  MoveL 7233 to (-64.74, 18.89, -264.72) mm, rotated rx 105.8 ry 33.04 rz 34.05 deg; joints [-10.347, -22.359, 96.233, 141.056, 86.367, 19.409, -475]
  MoveL 7234 to (-64.97, 19.26, -264.23) mm, rotated rx 105.8 ry 33.04 rz 34.05 deg; joints [-10.328, -22.332, 96.216, 141.075, 86.371, 19.399, -475]
  MoveL 7235 to (-64.83, 18.38, -263.37) mm, rotated rx 105.8 ry 33.04 rz 34.05 deg; joints [-10.295, -22.38, 96.234, 141.106, 86.342, 19.41, -475]
  MoveL 7236 to (-64.29, 14.15, -263.37) mm, rotated rx 105.8 ry 33.04 rz 34.05 deg; joints [-10.289, -22.594, 96.267, 141.105, 86.2, 19.523, -475]
  MoveL 7237 to (-64.04, 12.17, -263.31) mm, rotated rx 105.8 ry 33.04 rz 34.05 deg; joints [-10.284, -22.694, 96.282, 141.106, 86.132, 19.576, -475]
  MoveL 7238 to (-63.81, 10.19, -263.16) mm, rotated rx 105.8 ry 33.04 rz 34.05 deg; joints [-10.275, -22.794, 96.296, 141.111, 86.064, 19.628, -475]
  MoveL 7239 to (-63.54, 7.91, -262.96) mm, rotated rx 105.8 ry 33.04 rz 34.05 deg; joints [-10.264, -22.908, 96.312, 141.117, 85.986, 19.687, -475]
  MoveL 7240 to (-63.28, 5.75, -262.75) mm, rotated rx 105.8 ry 33.04 rz 34.05 deg; joints [-10.253, -23.016, 96.327, 141.124, 85.912, 19.743, -475]
  MoveL 7241 to (-63.02, 3.59, -262.65) mm, rotated rx 105.8 ry 33.04 rz 34.05 deg; joints [-10.246, -23.125, 96.342, 141.126, 85.837, 19.8, -475]
  MoveL 7242 to (-62.75, 1.47, -262.65) mm, rotated rx 105.8 ry 33.04 rz 34.05 deg; joints [-10.243, -23.231, 96.356, 141.125, 85.765, 19.858, -475]
  MoveL 7243 to (-62.49, -0.5, -262.58) mm, rotated rx 105.8 ry 33.04 rz 34.05 deg; joints [-10.238, -23.33, 96.37, 141.126, 85.698, 19.91, -475]
  MoveL 7244 to (-62.25, -2.36, -262.47) mm, rotated rx 105.8 ry 33.04 rz 34.05 deg; joints [-10.231, -23.423, 96.383, 141.129, 85.634, 19.959, -475]
  MoveL 7245 to (-61.99, -4.38, -262.4) mm, rotated rx 105.8 ry 33.04 rz 34.05 deg; joints [-10.226, -23.525, 96.396, 141.13, 85.564, 20.014, -475]
  MoveL 7246 to (-61.72, -6.5, -262.22) mm, rotated rx 105.8 ry 33.04 rz 34.05 deg; joints [-10.216, -23.631, 96.411, 141.135, 85.491, 20.069, -475]
  MoveL 7247 to (-61.18, -10.73, -262.04) mm, rotated rx 105.8 ry 33.04 rz 34.05 deg; joints [-10.203, -23.842, 96.437, 141.138, 85.345, 20.182, -475]
  MoveL 7248 to (-60.89, -12.85, -261.86) mm, rotated rx 105.8 ry 33.04 rz 34.05 deg; joints [-10.193, -23.949, 96.451, 141.143, 85.271, 20.238, -475]
  MoveL 7249 to (-60.61, -14.97, -261.68) mm, rotated rx 105.8 ry 33.04 rz 34.05 deg; joints [-10.184, -24.055, 96.466, 141.148, 85.198, 20.293, -475]
  MoveL 7250 to (-60.34, -17.08, -261.68) mm, rotated rx 105.8 ry 33.04 rz 34.05 deg; joints [-10.181, -24.16, 96.477, 141.145, 85.124, 20.352, -475]
  MoveL 7251 to (-60.05, -19.2, -261.5) mm, rotated rx 105.8 ry 33.04 rz 34.05 deg; joints [-10.171, -24.266, 96.491, 141.15, 85.051, 20.408, -475]
  MoveL 7252 to (-59.75, -21.31, -261.32) mm, rotated rx 105.8 ry 33.04 rz 34.05 deg; joints [-10.162, -24.372, 96.505, 141.154, 84.977, 20.463, -475]
  MoveL 7253 to (-59.48, -23.43, -261.32) mm, rotated rx 105.8 ry 33.04 rz 34.05 deg; joints [-10.159, -24.476, 96.515, 141.152, 84.903, 20.522, -475]
  MoveL 7254 to (-59.16, -25.35, -261.13) mm, rotated rx 105.8 ry 33.04 rz 34.05 deg; joints [-10.149, -24.575, 96.532, 141.157, 84.838, 20.571, -475]
  MoveL 7255 to (-58.82, -27.03, -260.81) mm, rotated rx 105.8 ry 33.04 rz 34.05 deg; joints [-10.135, -24.665, 96.555, 141.166, 84.783, 20.61, -475]
  MoveL 7256 to (-58.43, -28.51, -260.34) mm, rotated rx 105.8 ry 33.04 rz 34.05 deg; joints [-10.116, -24.75, 96.585, 141.182, 84.737, 20.639, -475]
  MoveL 7257 to (-58.38, -27.56, -259.58) mm, rotated rx 105.8 ry 33.04 rz 34.05 deg; joints [-10.089, -24.714, 96.605, 141.211, 84.775, 20.598, -475]
  MoveL 7258 to (-58.37, -27.98, -259.57) mm, rotated rx 105.8 ry 33.04 rz 34.05 deg; joints [-10.088, -24.732, 96.603, 141.211, 84.758, 20.611, -475]
  MoveC 7259 to (-59.7, -31.27, -259.57) mm, rotated rx 105.8 ry 33.04 rz 34.05 deg; joints [-10.078, -24.802, 96.443, 141.207, 84.578, 20.752, -475] to (-61.3, -34.45, -259.57) mm, rotated rx 105.8 ry 33.04 rz 34.05 deg; joints [-10.067, -24.851, 96.257, 141.203, 84.392, 20.898, -475]
  MoveL 7260 to (-61.3, -34.45, -259.57) mm, rotated rx 105.8 ry 33.04 rz 34.05 deg; joints [-10.067, -24.851, 96.257, 141.203, 84.392, 20.898, -475]
  MoveL 7261 to (-61.5, -34.87, -259.55) mm, rotated rx 105.8 ry 33.04 rz 34.05 deg; joints [-10.065, -24.858, 96.234, 141.204, 84.368, 20.917, -475]
  MoveL 7262 to (-61.66, -35.26, -259.5) mm, rotated rx 105.8 ry 33.04 rz 34.05 deg; joints [-10.062, -24.866, 96.215, 141.205, 84.346, 20.933, -475]
  MoveL 7263 to (-61.81, -35.64, -259.44) mm, rotated rx 105.8 ry 33.04 rz 34.05 deg; joints [-10.058, -24.874, 96.197, 141.207, 84.326, 20.948, -475]
  MoveL 7264 to (-61.98, -36.04, -259.39) mm, rotated rx 105.8 ry 33.04 rz 34.05 deg; joints [-10.055, -24.882, 96.177, 141.208, 84.303, 20.965, -475]
  MoveL 7265 to (-62.18, -36.47, -259.36) mm, rotated rx 105.8 ry 33.04 rz 34.05 deg; joints [-10.053, -24.89, 96.153, 141.208, 84.278, 20.984, -475]
  MoveL 7266 to (-62.41, -36.94, -259.35) mm, rotated rx 105.8 ry 33.04 rz 34.05 deg; joints [-10.051, -24.897, 96.127, 141.208, 84.251, 21.005, -475]
  MoveL 7267 to (-62.87, -37.88, -259.35) mm, rotated rx 105.8 ry 33.04 rz 34.05 deg; joints [-10.048, -24.912, 96.072, 141.207, 84.197, 21.048, -475]
  MoveL 7268 to (-63.58, -39.15, -259.44) mm, rotated rx 105.8 ry 33.04 rz 34.05 deg; joints [-10.047, -24.928, 95.99, 141.202, 84.12, 21.109, -475]
  MoveL 7269 to (-64.26, -40.14, -259.71) mm, rotated rx 105.8 ry 33.04 rz 34.05 deg; joints [-10.053, -24.931, 95.91, 141.19, 84.056, 21.164, -475]
  MoveL 7270 to (-64.93, -40.84, -260.17) mm, rotated rx 105.8 ry 33.04 rz 34.05 deg; joints [-10.067, -24.924, 95.833, 141.172, 84.005, 21.211, -475]
  MoveL 7271 to (-65.58, -41.24, -260.81) mm, rotated rx 105.8 ry 33.04 rz 34.05 deg; joints [-10.088, -24.904, 95.759, 141.148, 83.967, 21.251, -475]
  MoveL 7272 to (-66.22, -41.37, -261.63) mm, rotated rx 105.8 ry 33.04 rz 34.05 deg; joints [-10.116, -24.873, 95.687, 141.118, 83.941, 21.284, -475]
  MoveL 7273 to (-66.84, -41.2, -262.64) mm, rotated rx 105.8 ry 33.04 rz 34.05 deg; joints [-10.152, -24.831, 95.618, 141.081, 83.928, 21.31, -475]
  MoveL 7274 to (-68.03, -40, -265.2) mm, rotated rx 105.8 ry 33.04 rz 34.05 deg; joints [-10.246, -24.711, 95.488, 140.989, 83.939, 21.34, -475]
  MoveL 7275 to (-68.83, -38.11, -267.76) mm, rotated rx 105.8 ry 33.04 rz 34.05 deg; joints [-10.342, -24.583, 95.402, 140.899, 83.992, 21.338, -475]
  MoveL 7276 to (-68.96, -37.08, -268.76) mm, rotated rx 105.8 ry 33.04 rz 34.05 deg; joints [-10.381, -24.53, 95.389, 140.863, 84.031, 21.323, -475]
  MoveL 7277 to (-68.91, -35.99, -269.59) mm, rotated rx 105.8 ry 33.04 rz 34.05 deg; joints [-10.414, -24.486, 95.397, 140.835, 84.078, 21.299, -475]
  MoveL 7278 to (-68.68, -34.85, -270.23) mm, rotated rx 105.8 ry 33.04 rz 34.05 deg; joints [-10.441, -24.449, 95.424, 140.813, 84.133, 21.265, -475]
  MoveL 7279 to (-68.27, -33.66, -270.68) mm, rotated rx 105.8 ry 33.04 rz 34.05 deg; joints [-10.461, -24.42, 95.471, 140.798, 84.196, 21.221, -475]
  MoveL 7280 to (-66.91, -31.1, -271.05) mm, rotated rx 105.8 ry 33.04 rz 34.05 deg; joints [-10.484, -24.384, 95.625, 140.788, 84.349, 21.106, -475]
  MoveL 7281 to (-66.34, -30.22, -271.05) mm, rotated rx 105.8 ry 33.04 rz 34.05 deg; joints [-10.488, -24.377, 95.689, 140.789, 84.404, 21.062, -475]
  MoveL 7282 to (-66.06, -29.78, -271.06) mm, rotated rx 105.8 ry 33.04 rz 34.05 deg; joints [-10.49, -24.373, 95.721, 140.789, 84.432, 21.04, -475]
  MoveL 7283 to (-65.81, -29.37, -271.08) mm, rotated rx 105.8 ry 33.04 rz 34.05 deg; joints [-10.493, -24.369, 95.749, 140.788, 84.457, 21.021, -475]
  MoveL 7284 to (-65.6, -29, -271.13) mm, rotated rx 105.8 ry 33.04 rz 34.05 deg; joints [-10.496, -24.364, 95.772, 140.787, 84.48, 21.004, -475]
  MoveL 7285 to (-65.41, -28.65, -271.18) mm, rotated rx 105.8 ry 33.04 rz 34.05 deg; joints [-10.499, -24.359, 95.793, 140.785, 84.501, 20.988, -475]
  MoveL 7286 to (-65.21, -28.28, -271.23) mm, rotated rx 105.8 ry 33.04 rz 34.05 deg; joints [-10.502, -24.354, 95.816, 140.784, 84.523, 20.971, -475]
  MoveL 7287 to (-64.96, -27.88, -271.25) mm, rotated rx 105.8 ry 33.04 rz 34.05 deg; joints [-10.505, -24.35, 95.844, 140.783, 84.548, 20.952, -475]
  MoveL 7288 to (-64.7, -27.46, -271.26) mm, rotated rx 105.8 ry 33.04 rz 34.05 deg; joints [-10.507, -24.347, 95.874, 140.783, 84.574, 20.931, -475]
  MoveL 7289 to (-64.4, -26.99, -271.25) mm, rotated rx 105.8 ry 33.04 rz 34.05 deg; joints [-10.508, -24.343, 95.908, 140.784, 84.604, 20.907, -475]
  MoveL 7290 to (-64.11, -26.55, -271.26) mm, rotated rx 105.8 ry 33.04 rz 34.05 deg; joints [-10.511, -24.339, 95.939, 140.784, 84.632, 20.885, -475]
  MoveL 7291 to (-63.85, -26.13, -271.28) mm, rotated rx 105.8 ry 33.04 rz 34.05 deg; joints [-10.513, -24.335, 95.968, 140.784, 84.658, 20.865, -475]
  MoveL 7292 to (-63.61, -25.72, -271.33) mm, rotated rx 105.8 ry 33.04 rz 34.05 deg; joints [-10.517, -24.33, 95.995, 140.782, 84.683, 20.845, -475]
  MoveL 7293 to (-63.37, -25.27, -271.41) mm, rotated rx 105.8 ry 33.04 rz 34.05 deg; joints [-10.521, -24.324, 96.022, 140.78, 84.709, 20.826, -475]
  MoveL 7294 to (-63.08, -24.74, -271.47) mm, rotated rx 105.8 ry 33.04 rz 34.05 deg; joints [-10.525, -24.317, 96.055, 140.778, 84.741, 20.801, -475]
  MoveL 7295 to (-62.78, -24.26, -271.49) mm, rotated rx 105.8 ry 33.04 rz 34.05 deg; joints [-10.528, -24.312, 96.088, 140.777, 84.771, 20.778, -475]
  MoveL 7296 to (-62.5, -23.81, -271.49) mm, rotated rx 105.8 ry 33.04 rz 34.05 deg; joints [-10.53, -24.308, 96.12, 140.778, 84.799, 20.755, -475]
  MoveL 7297 to (-62.21, -23.37, -271.49) mm, rotated rx 105.8 ry 33.04 rz 34.05 deg; joints [-10.532, -24.304, 96.151, 140.778, 84.827, 20.733, -475]
  MoveL 7298 to (-61.87, -22.81, -271.5) mm, rotated rx 105.8 ry 33.04 rz 34.05 deg; joints [-10.534, -24.298, 96.19, 140.778, 84.862, 20.706, -475]
  MoveL 7299 to (-61.59, -22.3, -271.51) mm, rotated rx 105.8 ry 33.04 rz 34.05 deg; joints [-10.537, -24.291, 96.222, 140.778, 84.893, 20.682, -475]
  MoveL 7300 to (-61.36, -21.85, -271.52) mm, rotated rx 105.8 ry 33.04 rz 34.05 deg; joints [-10.539, -24.284, 96.247, 140.778, 84.919, 20.661, -475]
  MoveL 7301 to (-61.26, -21.52, -271.52) mm, rotated rx 105.8 ry 33.04 rz 34.05 deg; joints [-10.54, -24.275, 96.26, 140.778, 84.935, 20.648, -475]
  MoveL 7302 to (-61.23, -21.25, -271.52) mm, rotated rx 105.8 ry 33.04 rz 34.05 deg; joints [-10.54, -24.266, 96.266, 140.778, 84.947, 20.638, -475]
  MoveL 7303 to (-61.34, -22.18, -272.11) mm, rotated rx 105.8 ry 33.04 rz 34.05 deg; joints [-10.56, -24.298, 96.241, 140.756, 84.907, 20.679, -475]
  MoveL 7304 to (-61.64, -20.88, -272.64) mm, rotated rx 105.8 ry 33.04 rz 34.05 deg; joints [-10.582, -24.225, 96.217, 140.738, 84.949, 20.654, -475]
  MoveL 7305 to (-61.85, -19.33, -273.02) mm, rotated rx 105.8 ry 33.04 rz 34.05 deg; joints [-10.598, -24.147, 96.205, 140.725, 85.003, 20.616, -475]
  MoveL 7306 to (-61.98, -17.49, -273.28) mm, rotated rx 105.8 ry 33.04 rz 34.05 deg; joints [-10.611, -24.061, 96.203, 140.717, 85.071, 20.565, -475]
  MoveL 7307 to (-62.05, -15.44, -273.41) mm, rotated rx 105.8 ry 33.04 rz 34.05 deg; joints [-10.62, -23.969, 96.211, 140.715, 85.149, 20.504, -475]
  MoveL 7308 to (-62.1, -13.33, -273.5) mm, rotated rx 105.8 ry 33.04 rz 34.05 deg; joints [-10.627, -23.876, 96.22, 140.713, 85.23, 20.441, -475]
  MoveL 7309 to (-62.2, -9.07, -273.68) mm, rotated rx 105.8 ry 33.04 rz 34.05 deg; joints [-10.641, -23.687, 96.239, 140.709, 85.394, 20.312, -475]
  MoveL 7310 to (-62.25, -6.94, -273.86) mm, rotated rx 105.8 ry 33.04 rz 34.05 deg; joints [-10.652, -23.592, 96.246, 140.704, 85.475, 20.249, -475]
  MoveL 7311 to (-62.34, -2.67, -274.04) mm, rotated rx 105.8 ry 33.04 rz 34.05 deg; joints [-10.667, -23.403, 96.264, 140.7, 85.638, 20.121, -475]
  MoveL 7312 to (-62.39, -0.54, -274.22) mm, rotated rx 105.8 ry 33.04 rz 34.05 deg; joints [-10.678, -23.307, 96.271, 140.694, 85.72, 20.058, -475]
  MoveL 7313 to (-62.43, 1.6, -274.31) mm, rotated rx 105.8 ry 33.04 rz 34.05 deg; joints [-10.685, -23.212, 96.279, 140.692, 85.801, 19.995, -475]
  MoveL 7314 to (-62.44, 3.57, -274.52) mm, rotated rx 105.8 ry 33.04 rz 34.05 deg; joints [-10.697, -23.125, 96.288, 140.685, 85.877, 19.936, -475]
  MoveL 7315 to (-62.48, 5.93, -274.67) mm, rotated rx 105.8 ry 33.04 rz 34.05 deg; joints [-10.707, -23.019, 96.296, 140.68, 85.967, 19.867, -475]
  MoveL 7316 to (-62.53, 8.49, -274.79) mm, rotated rx 105.8 ry 33.04 rz 34.05 deg; joints [-10.716, -22.904, 96.304, 140.677, 86.064, 19.79, -475]
  MoveL 7317 to (-62.57, 10.63, -274.79) mm, rotated rx 105.8 ry 33.04 rz 34.05 deg; joints [-10.72, -22.809, 96.312, 140.677, 86.145, 19.726, -475]
  MoveL 7318 to (-62.6, 12.66, -274.86) mm, rotated rx 105.8 ry 33.04 rz 34.05 deg; joints [-10.727, -22.718, 96.319, 140.675, 86.222, 19.665, -475]
  MoveL 7319 to (-62.61, 14.49, -275.04) mm, rotated rx 105.8 ry 33.04 rz 34.05 deg; joints [-10.737, -22.636, 96.325, 140.669, 86.292, 19.611, -475]
  MoveL 7320 to (-62.61, 16.36, -275.25) mm, rotated rx 105.8 ry 33.04 rz 34.05 deg; joints [-10.749, -22.553, 96.333, 140.661, 86.364, 19.556, -475]
  MoveL 7321 to (-62.64, 18.72, -275.38) mm, rotated rx 105.8 ry 33.04 rz 34.05 deg; joints [-10.759, -22.447, 96.34, 140.656, 86.453, 19.486, -475]
  MoveL 7322 to (-62.67, 21.3, -275.49) mm, rotated rx 105.8 ry 33.04 rz 34.05 deg; joints [-10.768, -22.33, 96.347, 140.652, 86.55, 19.41, -475]
  MoveL 7323 to (-62.75, 25.56, -275.49) mm, rotated rx 105.8 ry 33.04 rz 34.05 deg; joints [-10.776, -22.137, 96.358, 140.652, 86.71, 19.282, -475]
  MoveL 7324 to (-62.52, 25.78, -276.19) mm, rotated rx 105.8 ry 33.04 rz 34.05 deg; joints [-10.804, -22.137, 96.375, 140.625, 86.727, 19.277, -475]
  MoveL 7325 to (-62.39, 25.49, -276.53) mm, rotated rx 105.8 ry 33.04 rz 34.05 deg; joints [-10.817, -22.155, 96.383, 140.612, 86.722, 19.286, -475]
  MoveL 7326 to (-62.37, 25.49, -276.75) mm, rotated rx 105.8 ry 33.04 rz 34.05 deg; joints [-10.825, -22.156, 96.382, 140.604, 86.722, 19.288, -475]
  MoveL 7327 to (-62.46, 25.74, -276.86) mm, rotated rx 105.8 ry 33.04 rz 34.05 deg; joints [-10.829, -22.14, 96.373, 140.6, 86.729, 19.285, -475]
  MoveL 7328 to (-62.67, 26.14, -276.89) mm, rotated rx 105.8 ry 33.04 rz 34.05 deg; joints [-10.831, -22.111, 96.354, 140.599, 86.736, 19.279, -475]
  MoveL 7329 to (-62.91, 26.55, -276.92) mm, rotated rx 105.8 ry 33.04 rz 34.05 deg; joints [-10.831, -22.081, 96.331, 140.599, 86.742, 19.274, -475]
  MoveL 7330 to (-63.14, 26.92, -276.96) mm, rotated rx 105.8 ry 33.04 rz 34.05 deg; joints [-10.833, -22.053, 96.31, 140.597, 86.748, 19.27, -475]
  MoveL 7331 to (-63.34, 27.27, -277.03) mm, rotated rx 105.8 ry 33.04 rz 34.05 deg; joints [-10.836, -22.027, 96.291, 140.595, 86.753, 19.267, -475]
  MoveL 7332 to (-63.55, 27.62, -277.09) mm, rotated rx 105.8 ry 33.04 rz 34.05 deg; joints [-10.838, -22, 96.271, 140.593, 86.759, 19.263, -475]
  MoveL 7333 to (-63.79, 27.99, -277.13) mm, rotated rx 105.8 ry 33.04 rz 34.05 deg; joints [-10.839, -21.971, 96.248, 140.592, 86.764, 19.259, -475]
  MoveL 7334 to (-64.08, 28.43, -277.15) mm, rotated rx 105.8 ry 33.04 rz 34.05 deg; joints [-10.84, -21.937, 96.221, 140.592, 86.769, 19.255, -475]
  MoveL 7335 to (-64.36, 28.88, -277.22) mm, rotated rx 105.8 ry 33.04 rz 34.05 deg; joints [-10.842, -21.903, 96.195, 140.59, 86.776, 19.25, -475]
  MoveL 7336 to (-64.64, 29.32, -277.25) mm, rotated rx 105.8 ry 33.04 rz 34.05 deg; joints [-10.843, -21.869, 96.168, 140.589, 86.782, 19.246, -475]
  MoveL 7337 to (-64.94, 29.75, -277.25) mm, rotated rx 105.8 ry 33.04 rz 34.05 deg; joints [-10.843, -21.835, 96.14, 140.589, 86.786, 19.242, -475]
  MoveL 7338 to (-65.24, 30.18, -277.25) mm, rotated rx 105.8 ry 33.04 rz 34.05 deg; joints [-10.843, -21.8, 96.112, 140.59, 86.791, 19.238, -475]
  MoveL 7339 to (-65.64, 30.73, -277.22) mm, rotated rx 105.8 ry 33.04 rz 34.05 deg; joints [-10.841, -21.755, 96.074, 140.591, 86.797, 19.233, -475]
  MoveL 7340 to (-66.04, 31.27, -277.19) mm, rotated rx 105.8 ry 33.04 rz 34.05 deg; joints [-10.84, -21.711, 96.037, 140.593, 86.802, 19.228, -475]
  MoveL 7341 to (-66.38, 31.76, -277.18) mm, rotated rx 105.8 ry 33.04 rz 34.05 deg; joints [-10.839, -21.672, 96.005, 140.594, 86.807, 19.224, -475]
  MoveL 7342 to (-66.63, 32.16, -277.22) mm, rotated rx 105.8 ry 33.04 rz 34.05 deg; joints [-10.84, -21.641, 95.981, 140.593, 86.812, 19.22, -475]
  MoveL 7343 to (-66.84, 32.51, -277.28) mm, rotated rx 105.8 ry 33.04 rz 34.05 deg; joints [-10.843, -21.615, 95.961, 140.591, 86.818, 19.216, -475]
  MoveL 7344 to (-67.05, 32.86, -277.34) mm, rotated rx 105.8 ry 33.04 rz 34.05 deg; joints [-10.845, -21.588, 95.94, 140.589, 86.823, 19.213, -475]
  MoveL 7345 to (-67.29, 33.23, -277.37) mm, rotated rx 105.8 ry 33.04 rz 34.05 deg; joints [-10.846, -21.559, 95.918, 140.588, 86.828, 19.209, -475]
  MoveL 7346 to (-68.19, 34.52, -277.37) mm, rotated rx 105.8 ry 33.04 rz 34.05 deg; joints [-10.845, -21.456, 95.833, 140.59, 86.842, 19.197, -475]
  MoveL 7347 to (-69.65, 37.02, -277.75) mm, rotated rx 105.8 ry 33.04 rz 34.05 deg; joints [-10.859, -21.27, 95.692, 140.578, 86.879, 19.171, -475]
  MoveL 7348 to (-70.11, 38.18, -278.22) mm, rotated rx 105.8 ry 33.04 rz 34.05 deg; joints [-10.877, -21.193, 95.645, 140.561, 86.905, 19.156, -475]
  MoveL 7349 to (-70.4, 39.29, -278.88) mm, rotated rx 105.8 ry 33.04 rz 34.05 deg; joints [-10.903, -21.127, 95.613, 140.537, 86.936, 19.14, -475]
  MoveL 7350 to (-70.51, 40.34, -279.72) mm, rotated rx 105.8 ry 33.04 rz 34.05 deg; joints [-10.937, -21.072, 95.597, 140.505, 86.972, 19.122, -475]
  MoveL 7351 to (-70.44, 41.34, -280.76) mm, rotated rx 105.8 ry 33.04 rz 34.05 deg; joints [-10.979, -21.028, 95.596, 140.466, 87.012, 19.103, -475]
  MoveL 7352 to (-69.77, 43.17, -283.4) mm, rotated rx 105.8 ry 33.04 rz 34.05 deg; joints [-11.085, -20.973, 95.641, 140.365, 87.107, 19.061, -475]
  MoveL 7353 to (-68.68, 44.33, -286.03) mm, rotated rx 105.8 ry 33.04 rz 34.05 deg; joints [-11.192, -20.968, 95.725, 140.264, 87.194, 19.026, -475]
  MoveL 7354 to (-68.09, 44.48, -287.07) mm, rotated rx 105.8 ry 33.04 rz 34.05 deg; joints [-11.234, -20.988, 95.774, 140.224, 87.223, 19.016, -475]
  MoveL 7355 to (-67.46, 44.36, -287.92) mm, rotated rx 105.8 ry 33.04 rz 34.05 deg; joints [-11.268, -21.023, 95.827, 140.191, 87.243, 19.011, -475]
  MoveL 7356 to (-66.81, 43.95, -288.58) mm, rotated rx 105.8 ry 33.04 rz 34.05 deg; joints [-11.295, -21.073, 95.884, 140.165, 87.253, 19.012, -475]
  MoveL 7357 to (-66.12, 43.27, -289.05) mm, rotated rx 105.8 ry 33.04 rz 34.05 deg; joints [-11.314, -21.137, 95.946, 140.147, 87.254, 19.017, -475]
  MoveL 7358 to (-65.39, 42.3, -289.33) mm, rotated rx 105.8 ry 33.04 rz 34.05 deg; joints [-11.326, -21.216, 96.012, 140.135, 87.246, 19.028, -475]
  MoveL 7359 to (-64.64, 41.05, -289.42) mm, rotated rx 105.8 ry 33.04 rz 34.05 deg; joints [-11.33, -21.31, 96.082, 140.13, 87.229, 19.044, -475]
  MoveL 7360 to (-64.38, 40.6, -289.42) mm, rotated rx 105.8 ry 33.04 rz 34.05 deg; joints [-11.33, -21.343, 96.106, 140.13, 87.222, 19.05, -475]
  MoveL 7361 to (-64.17, 40.18, -289.4) mm, rotated rx 105.8 ry 33.04 rz 34.05 deg; joints [-11.329, -21.373, 96.127, 140.13, 87.215, 19.055, -475]
  MoveL 7362 to (-63.99, 39.82, -289.36) mm, rotated rx 105.8 ry 33.04 rz 34.05 deg; joints [-11.327, -21.398, 96.143, 140.132, 87.208, 19.061, -475]
  MoveL 7363 to (-63.83, 39.46, -289.3) mm, rotated rx 105.8 ry 33.04 rz 34.05 deg; joints [-11.325, -21.423, 96.159, 140.134, 87.201, 19.066, -475]
  MoveL 7364 to (-63.64, 39.07, -289.26) mm, rotated rx 105.8 ry 33.04 rz 34.05 deg; joints [-11.323, -21.45, 96.177, 140.135, 87.193, 19.071, -475]
  MoveL 7365 to (-63.41, 38.64, -289.23) mm, rotated rx 105.8 ry 33.04 rz 34.05 deg; joints [-11.322, -21.481, 96.199, 140.136, 87.186, 19.077, -475]
  MoveL 7366 to (-63.16, 38.18, -289.23) mm, rotated rx 105.8 ry 33.04 rz 34.05 deg; joints [-11.322, -21.514, 96.222, 140.136, 87.178, 19.083, -475]
  MoveL 7367 to (-62.94, 37.77, -289.21) mm, rotated rx 105.8 ry 33.04 rz 34.05 deg; joints [-11.322, -21.544, 96.243, 140.136, 87.171, 19.089, -475]
  MoveL 7368 to (-62.76, 37.41, -289.16) mm, rotated rx 105.8 ry 33.04 rz 34.05 deg; joints [-11.319, -21.569, 96.261, 140.138, 87.165, 19.094, -475]
  MoveL 7369 to (-62.59, 37.06, -289.1) mm, rotated rx 105.8 ry 33.04 rz 34.05 deg; joints [-11.317, -21.594, 96.277, 140.14, 87.158, 19.098, -475]
  MoveL 7370 to (-62.39, 36.67, -289.05) mm, rotated rx 105.8 ry 33.04 rz 34.05 deg; joints [-11.315, -21.621, 96.296, 140.141, 87.151, 19.104, -475]
  MoveL 7371 to (-62.16, 36.24, -289.03) mm, rotated rx 105.8 ry 33.04 rz 34.05 deg; joints [-11.314, -21.652, 96.317, 140.142, 87.144, 19.109, -475]
  MoveL 7372 to (-61.91, 35.78, -289.03) mm, rotated rx 105.8 ry 33.04 rz 34.05 deg; joints [-11.314, -21.686, 96.341, 140.142, 87.137, 19.116, -475]
  MoveL 7373 to (-61.49, 34.89, -289.01) mm, rotated rx 105.8 ry 33.04 rz 34.05 deg; joints [-11.313, -21.747, 96.379, 140.142, 87.119, 19.13, -475]
  MoveC 7374 to (-60.95, 33.62, -289.01) mm, rotated rx 105.8 ry 33.04 rz 34.05 deg; joints [-11.313, -21.831, 96.429, 140.141, 87.092, 19.153, -475] to (-60.25, 32.43, -289.01) mm, rotated rx 105.8 ry 33.04 rz 34.05 deg; joints [-11.313, -21.92, 96.493, 140.14, 87.073, 19.168, -475]
  MoveL 7375 to (-60.25, 32.43, -289) mm, rotated rx 105.8 ry 33.04 rz 34.05 deg; joints [-11.313, -21.92, 96.493, 140.141, 87.073, 19.168, -475]
  MoveL 7376 to (-59.97, 31.83, -288.98) mm, rotated rx 105.8 ry 33.04 rz 34.05 deg; joints [-11.312, -21.961, 96.52, 140.141, 87.062, 19.177, -475]
  MoveL 7377 to (-59.78, 31.29, -288.96) mm, rotated rx 105.8 ry 33.04 rz 34.05 deg; joints [-11.311, -21.995, 96.537, 140.142, 87.049, 19.188, -475]
  MoveL 7378 to (-59.74, 30.99, -288.86) mm, rotated rx 105.8 ry 33.04 rz 34.05 deg; joints [-11.306, -22.011, 96.54, 140.145, 87.039, 19.195, -475]
  MoveL 7379 to (-59.8, 31.02, -288.66) mm, rotated rx 105.8 ry 33.04 rz 34.05 deg; joints [-11.299, -22.007, 96.537, 140.153, 87.038, 19.193, -475]
  MoveL 7380 to (-59.93, 31.42, -288.35) mm, rotated rx 105.8 ry 33.04 rz 34.05 deg; joints [-11.287, -21.983, 96.528, 140.164, 87.048, 19.181, -475]
  MoveL 7381 to (-60.3, 31.52, -287.73) mm, rotated rx 105.8 ry 33.04 rz 34.05 deg; joints [-11.263, -21.961, 96.499, 140.188, 87.037, 19.181, -475]
  MoveL 7382 to (-60.37, 29.49, -287.72) mm, rotated rx 105.8 ry 33.04 rz 34.05 deg; joints [-11.258, -22.049, 96.485, 140.19, 86.958, 19.245, -475]
  MoveL 7383 to (-60.52, 27.35, -287.67) mm, rotated rx 105.8 ry 33.04 rz 34.05 deg; joints [-11.25, -22.137, 96.462, 140.193, 86.872, 19.315, -475]
  MoveL 7384 to (-60.72, 25.09, -287.54) mm, rotated rx 105.8 ry 33.04 rz 34.05 deg; joints [-11.24, -22.228, 96.434, 140.199, 86.778, 19.389, -475]
  MoveL 7385 to (-60.92, 22.86, -287.44) mm, rotated rx 105.8 ry 33.04 rz 34.05 deg; joints [-11.231, -22.318, 96.406, 140.203, 86.686, 19.462, -475]
  MoveL 7386 to (-61.12, 20.72, -287.27) mm, rotated rx 105.8 ry 33.04 rz 34.05 deg; joints [-11.219, -22.403, 96.378, 140.211, 86.598, 19.532, -475]
  MoveL 7387 to (-61.3, 18.78, -287.12) mm, rotated rx 105.8 ry 33.04 rz 34.05 deg; joints [-11.209, -22.48, 96.353, 140.217, 86.517, 19.596, -475]
  MoveL 7388 to (-61.48, 16.72, -287.07) mm, rotated rx 105.8 ry 33.04 rz 34.05 deg; joints [-11.202, -22.562, 96.326, 140.219, 86.432, 19.664, -475]
  MoveL 7389 to (-61.67, 14.57, -287) mm, rotated rx 105.8 ry 33.04 rz 34.05 deg; joints [-11.194, -22.648, 96.298, 140.222, 86.343, 19.735, -475]
  MoveL 7390 to (-61.87, 12.23, -286.85) mm, rotated rx 105.8 ry 33.04 rz 34.05 deg; joints [-11.182, -22.741, 96.267, 140.228, 86.246, 19.812, -475]
  MoveL 7391 to (-62.04, 10.36, -286.73) mm, rotated rx 105.8 ry 33.04 rz 34.05 deg; joints [-11.174, -22.815, 96.242, 140.233, 86.168, 19.874, -475]
  MoveL 7392 to (-62.24, 7.98, -286.52) mm, rotated rx 105.8 ry 33.04 rz 34.05 deg; joints [-11.16, -22.91, 96.212, 140.241, 86.07, 19.951, -475]
  MoveL 7393 to (-62.39, 6.1, -286.41) mm, rotated rx 105.8 ry 33.04 rz 34.05 deg; joints [-11.151, -22.984, 96.187, 140.245, 85.992, 20.012, -475]
  MoveL 7394 to (-62.57, 3.98, -286.24) mm, rotated rx 105.8 ry 33.04 rz 34.05 deg; joints [-11.14, -23.068, 96.159, 140.251, 85.904, 20.082, -475]
  MoveL 7395 to (-62.76, 1.6, -286.19) mm, rotated rx 105.8 ry 33.04 rz 34.05 deg; joints [-11.132, -23.162, 96.126, 140.252, 85.805, 20.161, -475]
  MoveL 7396 to (-62.91, -0.28, -286.08) mm, rotated rx 105.8 ry 33.04 rz 34.05 deg; joints [-11.123, -23.236, 96.101, 140.256, 85.727, 20.223, -475]
  MoveL 7397 to (-63.08, -2.4, -285.92) mm, rotated rx 105.8 ry 33.04 rz 34.05 deg; joints [-11.112, -23.32, 96.073, 140.262, 85.639, 20.292, -475]
  MoveL 7398 to (-63.27, -4.78, -285.87) mm, rotated rx 105.8 ry 33.04 rz 34.05 deg; joints [-11.105, -23.413, 96.039, 140.263, 85.54, 20.372, -475]
  MoveL 7399 to (-63.42, -6.66, -285.75) mm, rotated rx 105.8 ry 33.04 rz 34.05 deg; joints [-11.096, -23.486, 96.013, 140.266, 85.462, 20.433, -475]
  MoveL 7400 to (-63.59, -8.87, -285.65) mm, rotated rx 105.8 ry 33.04 rz 34.05 deg; joints [-11.087, -23.573, 95.982, 140.269, 85.369, 20.507, -475]
  MoveL 7401 to (-63.76, -11.09, -285.58) mm, rotated rx 105.8 ry 33.04 rz 34.05 deg; joints [-11.079, -23.659, 95.95, 140.27, 85.277, 20.581, -475]
  MoveL 7402 to (-63.87, -12.97, -285.4) mm, rotated rx 105.8 ry 33.04 rz 34.05 deg; joints [-11.068, -23.734, 95.927, 140.276, 85.199, 20.641, -475]
  MoveL 7403 to (-63.95, -14.7, -285.15) mm, rotated rx 105.8 ry 33.04 rz 34.05 deg; joints [-11.055, -23.805, 95.909, 140.284, 85.129, 20.695, -475]
  MoveL 7404 to (-64, -16.32, -284.8) mm, rotated rx 105.8 ry 33.04 rz 34.05 deg; joints [-11.038, -23.873, 95.897, 140.296, 85.063, 20.742, -475]
  MoveL 7405 to (-63.46, -14.92, -284.11) mm, rotated rx 105.8 ry 33.04 rz 34.05 deg; joints [-11.017, -23.843, 95.968, 140.321, 85.137, 20.673, -475]
  MoveL 7406 to (-63.52, -15.14, -284.1) mm, rotated rx 105.8 ry 33.04 rz 34.05 deg; joints [-11.017, -23.85, 95.96, 140.321, 85.126, 20.681, -475]
  MoveL 7407 to (-63.63, -15.41, -284.09) mm, rotated rx 105.8 ry 33.04 rz 34.05 deg; joints [-11.015, -23.855, 95.947, 140.322, 85.111, 20.693, -475]
  MoveL 7408 to (-63.87, -15.8, -284.06) mm, rotated rx 105.8 ry 33.04 rz 34.05 deg; joints [-11.012, -23.859, 95.92, 140.323, 85.087, 20.712, -475]
  MoveL 7409 to (-64.18, -16.25, -284.02) mm, rotated rx 105.8 ry 33.04 rz 34.05 deg; joints [-11.009, -23.863, 95.888, 140.324, 85.058, 20.735, -475]
  MoveL 7410 to (-64.54, -16.74, -283.98) mm, rotated rx 105.8 ry 33.04 rz 34.05 deg; joints [-11.005, -23.865, 95.848, 140.326, 85.026, 20.76, -475]
  MoveL 7411 to (-66.17, -18.79, -283.98) mm, rotated rx 105.8 ry 33.04 rz 34.05 deg; joints [-10.994, -23.866, 95.67, 140.326, 84.886, 20.873, -475]
  MoveL 7412 to (-66.54, -19.28, -283.95) mm, rotated rx 105.8 ry 33.04 rz 34.05 deg; joints [-10.991, -23.868, 95.631, 140.327, 84.853, 20.898, -475]
  MoveL 7413 to (-66.94, -19.83, -283.89) mm, rotated rx 105.8 ry 33.04 rz 34.05 deg; joints [-10.986, -23.87, 95.587, 140.329, 84.817, 20.927, -475]
  MoveL 7414 to (-67.32, -20.33, -283.86) mm, rotated rx 105.8 ry 33.04 rz 34.05 deg; joints [-10.983, -23.872, 95.546, 140.33, 84.783, 20.953, -475]
  MoveL 7415 to (-67.65, -20.74, -283.86) mm, rotated rx 105.8 ry 33.04 rz 34.05 deg; joints [-10.981, -23.872, 95.51, 140.33, 84.755, 20.976, -475]
  MoveL 7416 to (-67.95, -21.13, -283.85) mm, rotated rx 105.8 ry 33.04 rz 34.05 deg; joints [-10.978, -23.872, 95.476, 140.33, 84.729, 20.997, -475]
  MoveL 7417 to (-68.28, -21.53, -283.85) mm, rotated rx 105.8 ry 33.04 rz 34.05 deg; joints [-10.976, -23.872, 95.441, 140.33, 84.701, 21.019, -475]
  MoveL 7418 to (-68.6, -21.94, -283.85) mm, rotated rx 105.8 ry 33.04 rz 34.05 deg; joints [-10.974, -23.872, 95.406, 140.33, 84.673, 21.041, -475]
  MoveL 7419 to (-68.89, -22.32, -283.82) mm, rotated rx 105.8 ry 33.04 rz 34.05 deg; joints [-10.971, -23.873, 95.373, 140.331, 84.647, 21.062, -475]
  MoveL 7420 to (-69.17, -22.7, -283.77) mm, rotated rx 105.8 ry 33.04 rz 34.05 deg; joints [-10.968, -23.874, 95.344, 140.332, 84.623, 21.081, -475]
  MoveL 7421 to (-69.47, -23.09, -283.75) mm, rotated rx 105.8 ry 33.04 rz 34.05 deg; joints [-10.965, -23.875, 95.311, 140.333, 84.596, 21.102, -475]
  MoveL 7422 to (-69.8, -23.51, -283.75) mm, rotated rx 105.8 ry 33.04 rz 34.05 deg; joints [-10.963, -23.875, 95.274, 140.333, 84.568, 21.124, -475]
  MoveL 7423 to (-70.46, -24.32, -283.75) mm, rotated rx 105.8 ry 33.04 rz 34.05 deg; joints [-10.959, -23.875, 95.202, 140.332, 84.512, 21.169, -475]
  Set speed (1000.0 mm/s)
  MoveL 7424 to (-88.16, -36.72, -283.75) mm, rotated rx 105.8 ry 33.04 rz 34.05 deg; joints [-10.87, -23.44, 93.312, 140.32, 83.373, 22.081, -475]
  Set speed (1000.0 mm/s)
  MoveL 7425 to (-88.16, -36.72, -283.75) mm, rotated rx 105.8 ry 33.04 rz 34.05 deg; joints [-10.87, -23.44, 93.312, 140.32, 83.373, 22.081, -475]
